(* PLC project SafeLOGIC-1, BrAutomation SafeDESIGNER  4.2.0.17 *)
(* stored: companyURL http://www.br-automation.com, creationDateTime Thu Sep 22 17:12:08 2016 *)

PROGRAM DoorLock
  VAR  (* added by the conversion: wires and edge detectors of the diagram *)
    _OR33_OUT : BOOL;
  END_VAR

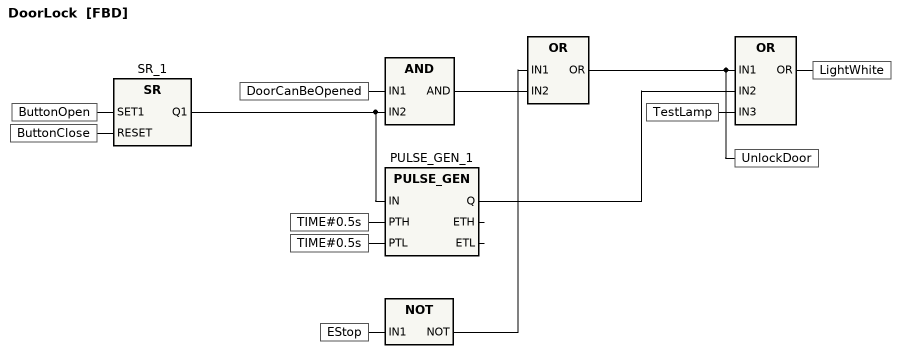
(* FBD diagram, written out as Structured Text *)
SR_1(SET1 := ButtonOpen, RESET := ButtonClose);
_OR33_OUT := NOT EStop OR DoorCanBeOpened AND SR_1.Q1;
UnlockDoor := _OR33_OUT;
PULSE_GEN_1(IN := SR_1.Q1, PTH := TIME#0.5s, PTL := TIME#0.5s);
LightWhite := _OR33_OUT OR PULSE_GEN_1.Q OR TestLamp;
END_PROGRAM
